(* Schneider Machine Expert - Basic project plc_prog_for_SoMachine_Basic, file version 2.2.0.0 *)
(* CompanyInformations: Name=SmallSystems *)
(* ProjectInformations: Name=Garden Water Control Centre, Description=Lorem ipsum dolor sit amet, consetetur sadipscing elitr, sed diam nonumy eirmod tempor invidunt ut labore et dolore magna aliquyam erat, sed diam voluptua. At vero eos et accusam et justo duo dolores et ea rebum. Stet clita kasd gubergren, no sea takimata sanctus est Lorem ipsum dolor sit amet. Lorem ipsum dolor sit amet, consetetur sadipscing elitr, sed diam nonumy eirmod tempor invidunt ut labore et dolore magna aliquyam erat, sed diam voluptua. At vero eos et accusam et justo duo dolores et ea rebum. Stet clita kasd gubergren, no sea takimata sanctus est Lorem ipsum dolor sit amet. *)
(* UserInformations: LastName=Wilhelm, FirstName=Konstantin, Email=admin@kw.smallsystems.ru, State=Brandenburg, Country=Germany *)

HARDWARE
  Cpu 0: TM221C16R
  EthernetConfiguration: NetworkName=M221, IpAllocationMode=FixedAddress, IpAddress=0.0.0.0, SubnetMask=0.0.0.0
  SerialLineConfiguration: Baud=Baud19200, Parity=ParityEven, DataBits=DataBits8, StopBits=StopBits1, PhysicalMedium=PhysicalMediumRs485, TransmissionMode=TransmissionModeModbusRtu, SlaveId=1, Addressing=SlaveAddressing
  MastTask: UsePeriodScanMode=false, PeriodScan=100
  FastTask: Period=255
  CpuBehavior: StartingMode=StartAsPreviousState, AutoSaveRamOnEeprom=true, WatchdogPeriod=250

SYMBOLS  (address, symbol, comment, settings)
  %M0       P_IN_RELEASE  "Freigabe für die Pumpe"
  %M1       P_IN_DELAY  "bei =1 darf die Pumpe NICHT AN sein"
  %M2       P_IN_TIMEOUT  "bei =1 muss die Pumpe ausgeschaltet sein"
  %M3       P_IN_OVERLOAD  "bei =1 muss die Pumpe ausgeschaltet sein"
  %M4       P_IN_OVERHEAT  "bei =1 muss die Pumpe ausgeschaltet sein"
  %M5       P_IN_BIT  "Merker, der das Status der Pumpe bestimmt"
  %M6       C_PIN_ERROR
  %M7       C_PIN_PRESET
  %M8       C_PIN_RESET
  %M9       C_PIN_SET
  %M10      C_PIN_CD
  %M11      P_OUT_RELEASE
  %M12      P_OUT_DELAY
  %M13      P_OUT_OVERLOAD
  %M14      P_OUT_OVERHEAT
  %M15      P_OUT_BIT
  %M16      P_OUT_TIMEOUT
  %M17      C_POUT_ERROR
  %M18      C_POUT_PRESET
  %M19      C_POUT_RESET
  %M20      C_POUT_SET
  %M21      C_POUT_CD
  %M22      VLV_TNK_UP_LEFT  "EINgangsventil im linken Behälter"
  %M23      VLV_TNK_UP_RIGHT  "EINgangsventil im rechten Behälter"
  %M24      VLV_IN_EXTENTION  "Zusätzlicher Vertil/Hand für Nebenanschluß an Pumpe_IN (Optional)"
  %M25      VLV_TNK_DOWN_LEFT  "AUSgangsventil im linken Behälter"
  %M26      VLV_TNK_DOWN_RIGHT  "AUSgangsventil im rechten Behälter"
  %M27      VLV_OUT_EXTENTION
  %M28      OUT_WITH_PRESSURE
  %M29      HIGH_LVL_TNK_LEFT  "Im linken Behälter hat das Wasser Höhepunk erreicht"
  %M30      HIGH_LVL_TNK_RIGHT  "Im linken Behälter hat das Wasser Höhepunk erreicht"
  %M31      LOW_LVL_TNK_LEFT
  %M32      LOW_LVL_TNK_RIGHT
  %M33      FILL_TNK_LEFT
  %M34      FILL_TNK_RIGHT
  %M35      DRAIN_TNK_LEFT
  %M36      DRAIN_TNK_RIGHT
  %S6       SB_TB1S  "Von einer internen Uhr generierte Zeitbasis 1 s"
  %S13      SB_FIRSTRUN  "Verweist auf den ersten Steuerungszyklus im RUN-Betrieb."
  %MW0      PUMP_DELAY_VALUE  "Die Stillzeit, die nach Ausschalten der Pumpe, eingehalten werden soll"
  %MW1      PUMP_TIMEOUT_VALUE  "Wie lange darf die Pumpe ununterbrochen laufen"
  %TM0      TP_P_IN  "Timer für die Pause zwischen EINschalten der Pumpe"  [Type=TP, Preset=120, Base=OneSecond]
  %TM1      TON_P_IN  "Timer für die maximale Dauer eines Einschltens"  [Preset=1200, Base=OneSecond]
  %TM2      TP_P_OUT  "Timer für die Pause zwischen EINschalten der Pumpe"  [Type=TP, Preset=120, Base=OneSecond]
  %TM3      TON_P_OUT  "Timer für die maximale Dauer eines Einschltens"  [Preset=1200, Base=OneSecond]
  %TM4        [Preset=10, Base=OneSecond]
  %TM5        [Preset=2, Base=OneSecond]
  %TM6        [Preset=2, Base=OneSecond]
  %TM7        [Preset=20, Base=OneSecond]
  %TM8        [Preset=20, Base=OneSecond]
  %TM9        [Preset=20, Base=OneSecond]
  %C0       COUNTER_P_IN  "Zählt die Arbeitszeit in Sekunden"  [Preset=7200]
  %C1       COUNTER_P_OUT  "Zählt die Arbeitszeit in Sekunden"  [Preset=7200]
  %I0.0     I_0_0
  %Q0.0     Q_0_0

POU IO
  (* SectionNumber=1 *)

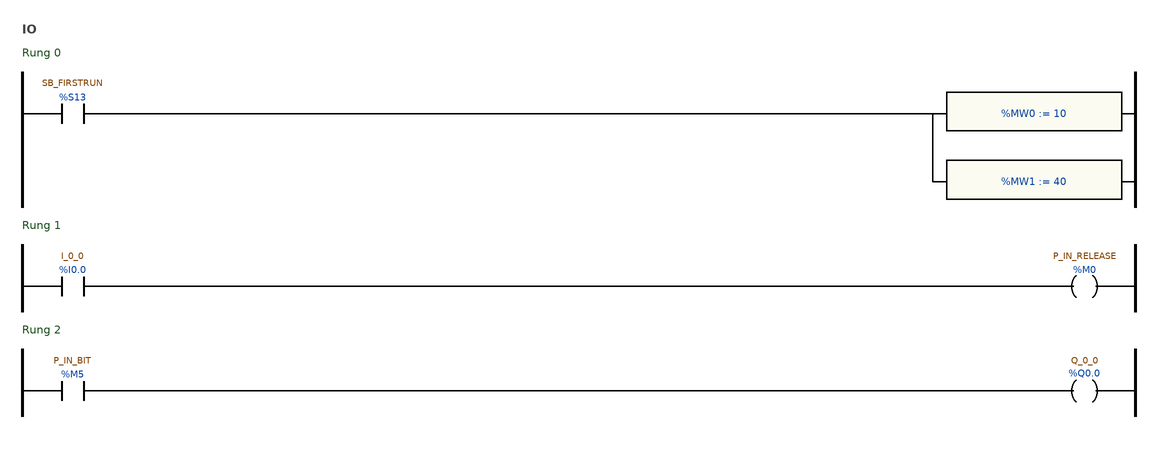

// Rung 0
  LD %S13                 (* SB_FIRSTRUN *)
  [ %MW0 := 10 ]          (* PUMP_DELAY_VALUE *)
  [ %MW1 := 40 ]          (* PUMP_TIMEOUT_VALUE *)
  // as ST:
  //   IF SB_FIRSTRUN THEN PUMP_DELAY_VALUE := 10; END_IF;
  //   IF SB_FIRSTRUN THEN PUMP_TIMEOUT_VALUE := 40; END_IF;

// Rung 1
  LD %I0.0                (* I_0_0 *)
  ST %M0                  (* P_IN_RELEASE *)
  // as ST:
  //   P_IN_RELEASE := I_0_0;

// Rung 2
  LD %M5                  (* P_IN_BIT *)
  ST %Q0.0                (* Q_0_0 *)
  // as ST:
  //   Q_0_0 := P_IN_BIT;

POU Valves
  (* SectionNumber=2 *)

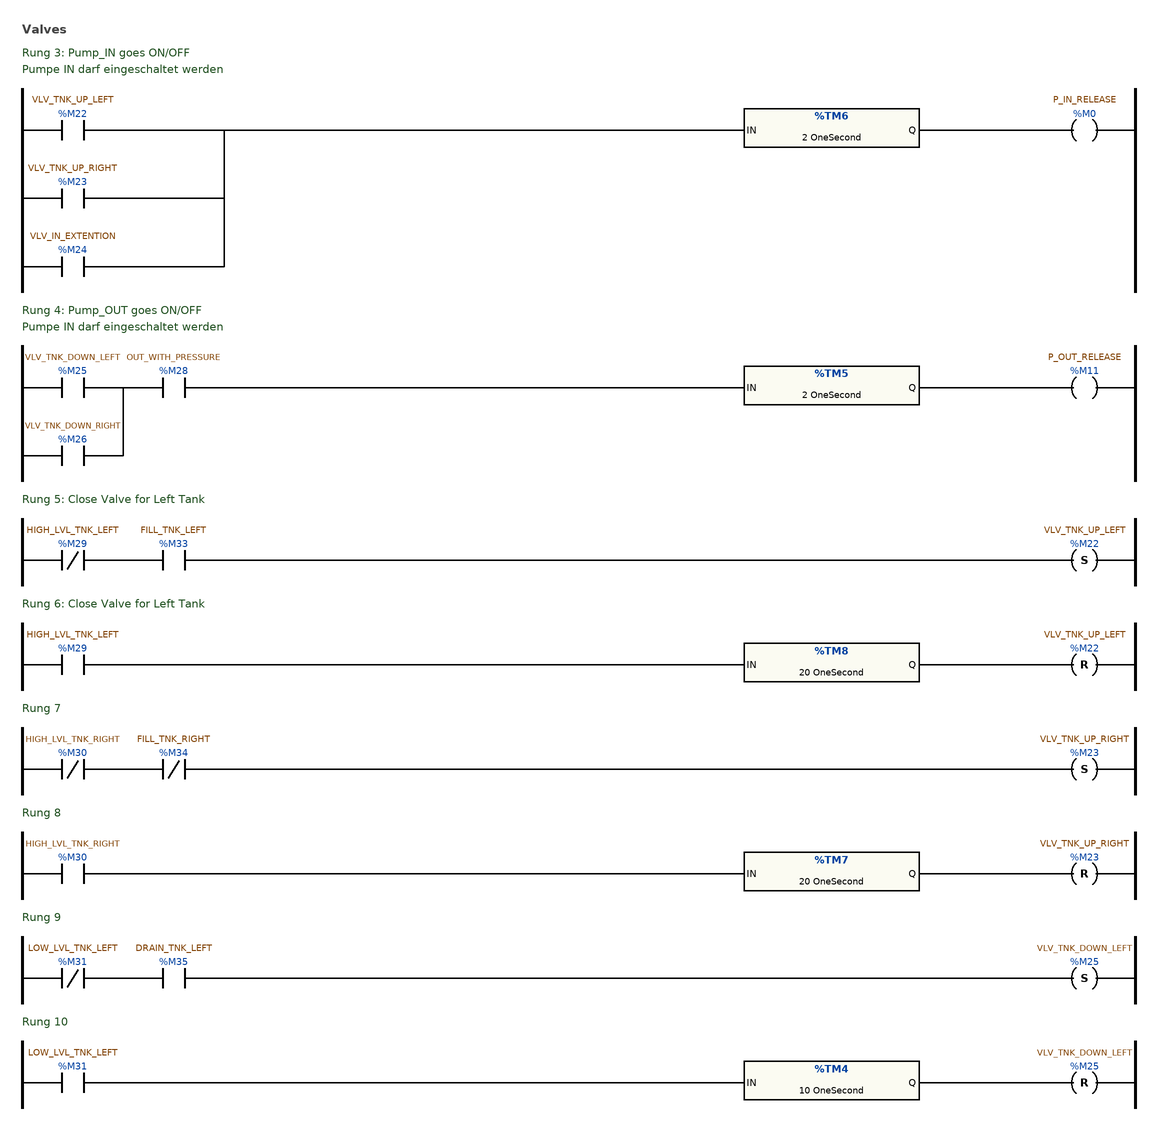

// Rung 3: Pump_IN goes ON/OFF
// Pumpe IN darf eingeschaltet werden
  BLK %TM6
  LD %M22                 (* VLV_TNK_UP_LEFT *)
  OR %M23                 (* VLV_TNK_UP_RIGHT *)
  OR %M24                 (* VLV_IN_EXTENTION *)
  IN
  OUT_BLK
  LD Q
  ST %M0                  (* P_IN_RELEASE *)
  END_BLK
  // as ST:
  //   %TM6(IN := VLV_TNK_UP_LEFT OR VLV_TNK_UP_RIGHT OR VLV_IN_EXTENTION);
  //   P_IN_RELEASE := %TM6.Q;

// Rung 4: Pump_OUT goes ON/OFF
// Pumpe IN darf eingeschaltet werden
  BLK %TM5
  LD %M25                 (* VLV_TNK_DOWN_LEFT *)
  OR %M26                 (* VLV_TNK_DOWN_RIGHT *)
  AND %M28                (* OUT_WITH_PRESSURE *)
  IN
  OUT_BLK
  LD Q
  ST %M11                 (* P_OUT_RELEASE *)
  END_BLK
  // as ST:
  //   %TM5(IN := (VLV_TNK_DOWN_LEFT OR VLV_TNK_DOWN_RIGHT) AND OUT_WITH_PRESSURE);
  //   P_OUT_RELEASE := %TM5.Q;

// Rung 5: Close Valve for Left Tank
  LDN %M29                (* HIGH_LVL_TNK_LEFT *)
  AND %M33                (* FILL_TNK_LEFT *)
  S %M22                  (* VLV_TNK_UP_LEFT *)
  // as ST:
  //   IF NOT HIGH_LVL_TNK_LEFT AND FILL_TNK_LEFT THEN VLV_TNK_UP_LEFT := TRUE; END_IF;

// Rung 6: Close Valve for Left Tank
  BLK %TM8
  LD %M29                 (* HIGH_LVL_TNK_LEFT *)
  IN
  OUT_BLK
  LD Q
  R %M22                  (* VLV_TNK_UP_LEFT *)
  END_BLK
  // as ST:
  //   %TM8(IN := HIGH_LVL_TNK_LEFT);
  //   IF %TM8.Q THEN VLV_TNK_UP_LEFT := FALSE; END_IF;

// Rung 7
  LDN %M30                (* HIGH_LVL_TNK_RIGHT *)
  ANDN %M34               (* FILL_TNK_RIGHT *)
  S %M23                  (* VLV_TNK_UP_RIGHT *)
  // as ST:
  //   IF NOT HIGH_LVL_TNK_RIGHT AND NOT FILL_TNK_RIGHT THEN VLV_TNK_UP_RIGHT := TRUE; END_IF;

// Rung 8
  BLK %TM7
  LD %M30                 (* HIGH_LVL_TNK_RIGHT *)
  IN
  OUT_BLK
  LD Q
  R %M23                  (* VLV_TNK_UP_RIGHT *)
  END_BLK
  // as ST:
  //   %TM7(IN := HIGH_LVL_TNK_RIGHT);
  //   IF %TM7.Q THEN VLV_TNK_UP_RIGHT := FALSE; END_IF;

// Rung 9
  LDN %M31                (* LOW_LVL_TNK_LEFT *)
  AND %M35                (* DRAIN_TNK_LEFT *)
  S %M25                  (* VLV_TNK_DOWN_LEFT *)
  // as ST:
  //   IF NOT LOW_LVL_TNK_LEFT AND DRAIN_TNK_LEFT THEN VLV_TNK_DOWN_LEFT := TRUE; END_IF;

// Rung 10
  BLK %TM4
  LD %M31                 (* LOW_LVL_TNK_LEFT *)
  IN
  OUT_BLK
  LD Q
  R %M25                  (* VLV_TNK_DOWN_LEFT *)
  END_BLK
  // as ST:
  //   %TM4(IN := LOW_LVL_TNK_LEFT);
  //   IF %TM4.Q THEN VLV_TNK_DOWN_LEFT := FALSE; END_IF;

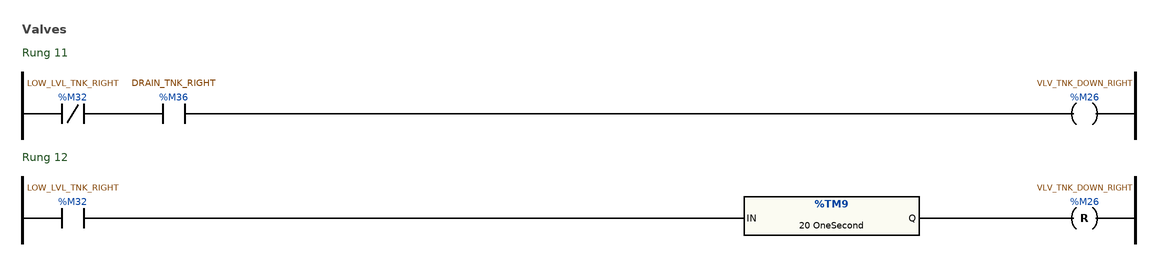

// Rung 11
  LDN %M32                (* LOW_LVL_TNK_RIGHT *)
  AND %M36                (* DRAIN_TNK_RIGHT *)
  ST %M26                 (* VLV_TNK_DOWN_RIGHT *)
  // as ST:
  //   VLV_TNK_DOWN_RIGHT := NOT LOW_LVL_TNK_RIGHT AND DRAIN_TNK_RIGHT;

// Rung 12
  BLK %TM9
  LD %M32                 (* LOW_LVL_TNK_RIGHT *)
  IN
  OUT_BLK
  LD Q
  R %M26                  (* VLV_TNK_DOWN_RIGHT *)
  END_BLK
  // as ST:
  //   %TM9(IN := LOW_LVL_TNK_RIGHT);
  //   IF %TM9.Q THEN VLV_TNK_DOWN_RIGHT := FALSE; END_IF;

POU Pumps
  (* SectionNumber=3 *)

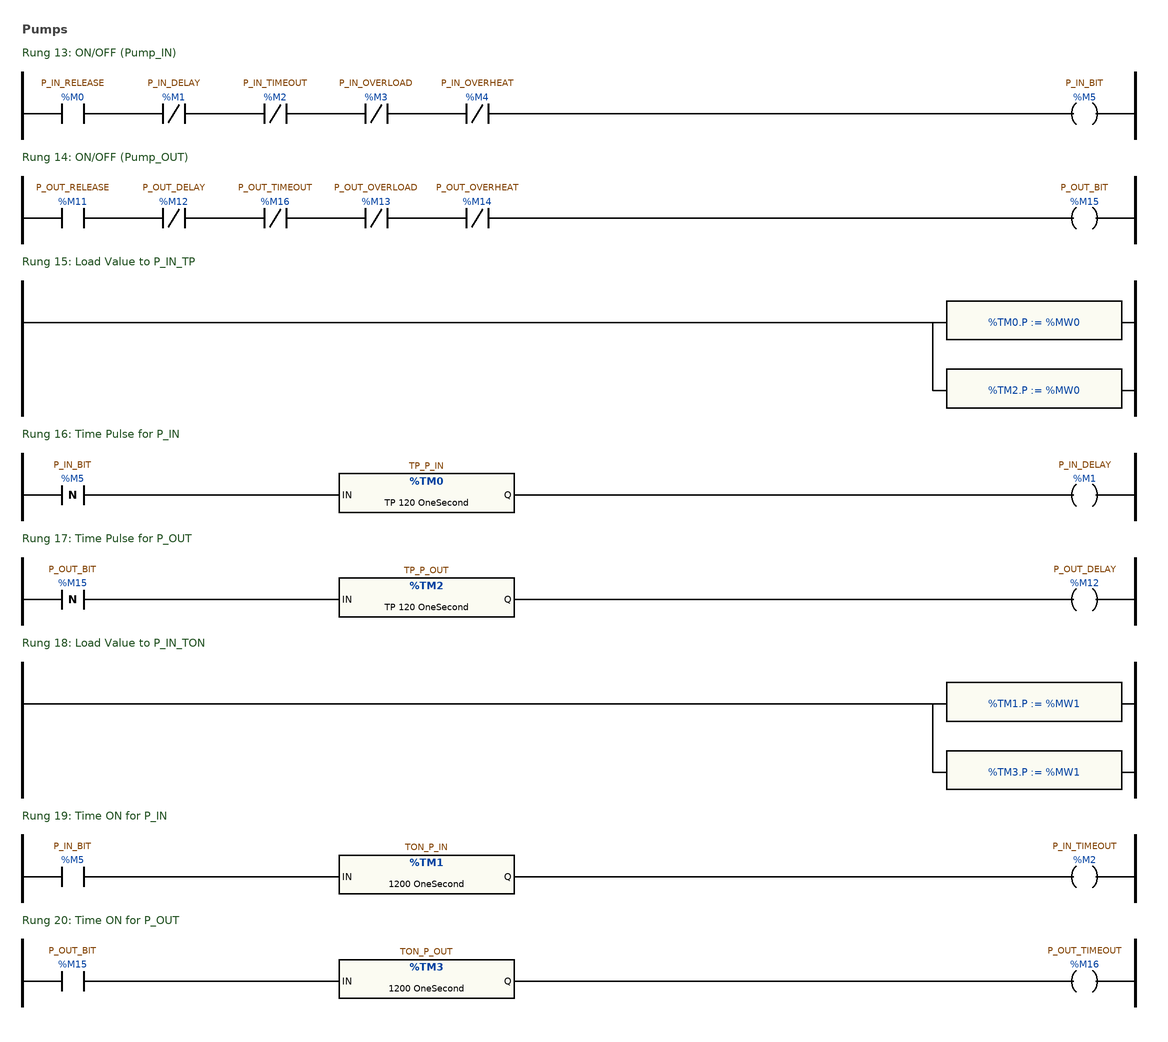

// Rung 13: ON/OFF (Pump_IN)
  LD %M0                  (* P_IN_RELEASE *)
  ANDN %M1                (* P_IN_DELAY *)
  ANDN %M2                (* P_IN_TIMEOUT *)
  ANDN %M3                (* P_IN_OVERLOAD *)
  ANDN %M4                (* P_IN_OVERHEAT *)
  ST %M5                  (* P_IN_BIT *)
  // as ST:
  //   P_IN_BIT := P_IN_RELEASE AND NOT P_IN_DELAY AND NOT P_IN_TIMEOUT AND NOT P_IN_OVERLOAD AND NOT P_IN_OVERHEAT;

// Rung 14: ON/OFF (Pump_OUT)
  LD %M11                 (* P_OUT_RELEASE *)
  ANDN %M12               (* P_OUT_DELAY *)
  ANDN %M16               (* P_OUT_TIMEOUT *)
  ANDN %M13               (* P_OUT_OVERLOAD *)
  ANDN %M14               (* P_OUT_OVERHEAT *)
  ST %M15                 (* P_OUT_BIT *)
  // as ST:
  //   P_OUT_BIT := P_OUT_RELEASE AND NOT P_OUT_DELAY AND NOT P_OUT_TIMEOUT AND NOT P_OUT_OVERLOAD AND NOT P_OUT_OVERHEAT;

// Rung 15: Load Value to P_IN_TP
  LD 1
  [ %TM0.P := %MW0 ]      (* TP_P_IN, PUMP_DELAY_VALUE - Laden Preset des Timers aus der Variable *)
  [ %TM2.P := %MW0 ]      (* TP_P_OUT, PUMP_DELAY_VALUE - Laden Preset des Timers aus der Variable *)
  // as ST:
  //   TP_P_IN.P := PUMP_DELAY_VALUE;
  //   TP_P_OUT.P := PUMP_DELAY_VALUE;

// Rung 16: Time Pulse for P_IN
  BLK %TM0                (* TP_P_IN *)
  LDF %M5                 (* P_IN_BIT *)
  IN
  OUT_BLK
  LD Q
  ST %M1                  (* P_IN_DELAY *)
  END_BLK
  // as ST:
  //   TP_P_IN(IN := FALLING(P_IN_BIT));
  //   P_IN_DELAY := TP_P_IN.Q;

// Rung 17: Time Pulse for P_OUT
  BLK %TM2                (* TP_P_OUT *)
  LDF %M15                (* P_OUT_BIT *)
  IN
  OUT_BLK
  LD Q
  ST %M12                 (* P_OUT_DELAY *)
  END_BLK
  // as ST:
  //   TP_P_OUT(IN := FALLING(P_OUT_BIT));
  //   P_OUT_DELAY := TP_P_OUT.Q;

// Rung 18: Load Value to P_IN_TON
  LD 1
  [ %TM1.P := %MW1 ]      (* TON_P_IN, PUMP_TIMEOUT_VALUE - Laden Preset des Timers aus der Variable *)
  [ %TM3.P := %MW1 ]      (* TON_P_OUT, PUMP_TIMEOUT_VALUE - Laden Preset des Timers aus der Variable *)
  // as ST:
  //   TON_P_IN.P := PUMP_TIMEOUT_VALUE;
  //   TON_P_OUT.P := PUMP_TIMEOUT_VALUE;

// Rung 19: Time ON for P_IN
  BLK %TM1                (* TON_P_IN *)
  LD %M5                  (* P_IN_BIT *)
  IN
  OUT_BLK
  LD Q
  ST %M2                  (* P_IN_TIMEOUT *)
  END_BLK
  // as ST:
  //   TON_P_IN(IN := P_IN_BIT);
  //   P_IN_TIMEOUT := TON_P_IN.Q;

// Rung 20: Time ON for P_OUT
  BLK %TM3                (* TON_P_OUT *)
  LD %M15                 (* P_OUT_BIT *)
  IN
  OUT_BLK
  LD Q
  ST %M16                 (* P_OUT_TIMEOUT *)
  END_BLK
  // as ST:
  //   TON_P_OUT(IN := P_OUT_BIT);
  //   P_OUT_TIMEOUT := TON_P_OUT.Q;

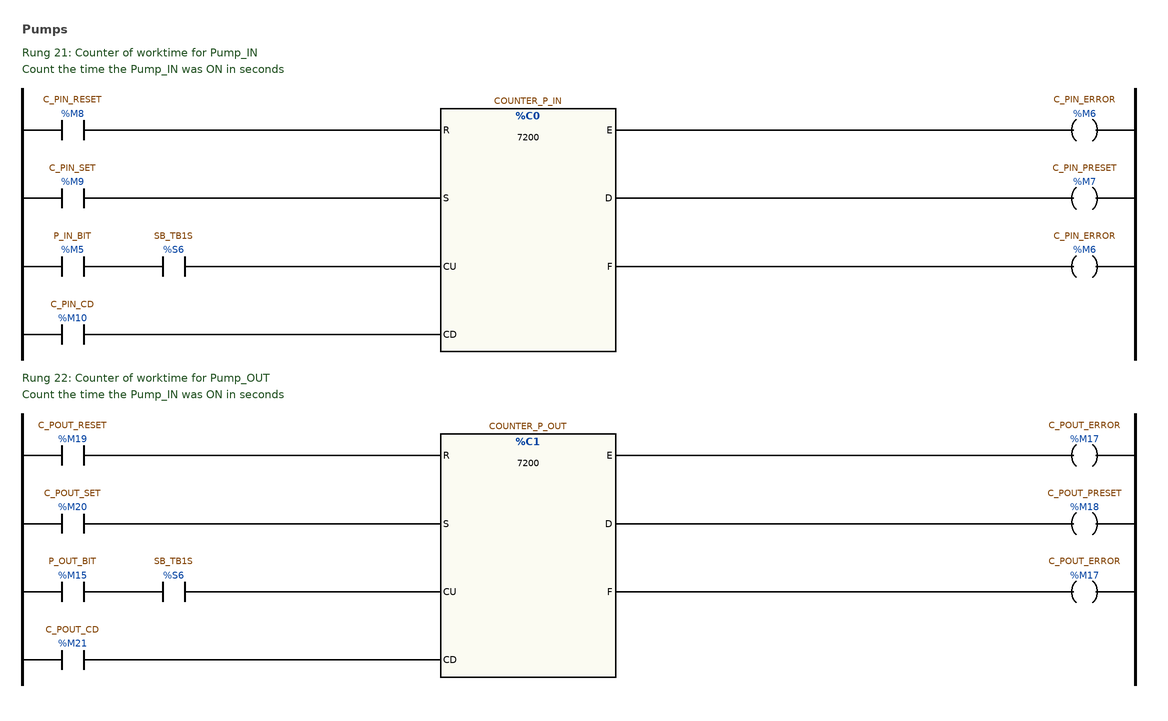

// Rung 21: Counter of worktime for Pump_IN
// Count the time the Pump_IN was ON in seconds
  BLK %C0                 (* COUNTER_P_IN *)
  LD %M8                  (* C_PIN_RESET *)
  R
  LD %M9                  (* C_PIN_SET *)
  S
  LD %M5                  (* P_IN_BIT *)
  AND %S6                 (* SB_TB1S *)
  CU
  LD %M10                 (* C_PIN_CD *)
  CD
  OUT_BLK
  LD E
  ST %M6                  (* C_PIN_ERROR *)
  LD D
  ST %M7                  (* C_PIN_PRESET *)
  LD F
  ST %M6                  (* C_PIN_ERROR *)
  END_BLK
  // as ST:
  //   COUNTER_P_IN(R := C_PIN_RESET, S := C_PIN_SET, CU := P_IN_BIT AND SB_TB1S, CD := C_PIN_CD);
  //   C_PIN_ERROR := COUNTER_P_IN.E;
  //   C_PIN_PRESET := COUNTER_P_IN.D;
  //   C_PIN_ERROR := COUNTER_P_IN.F;

// Rung 22: Counter of worktime for Pump_OUT
// Count the time the Pump_IN was ON in seconds
  BLK %C1                 (* COUNTER_P_OUT *)
  LD %M19                 (* C_POUT_RESET *)
  R
  LD %M20                 (* C_POUT_SET *)
  S
  LD %M15                 (* P_OUT_BIT *)
  AND %S6                 (* SB_TB1S *)
  CU
  LD %M21                 (* C_POUT_CD *)
  CD
  OUT_BLK
  LD E
  ST %M17                 (* C_POUT_ERROR *)
  LD D
  ST %M18                 (* C_POUT_PRESET *)
  LD F
  ST %M17                 (* C_POUT_ERROR *)
  END_BLK
  // as ST:
  //   COUNTER_P_OUT(R := C_POUT_RESET, S := C_POUT_SET, CU := P_OUT_BIT AND SB_TB1S, CD := C_POUT_CD);
  //   C_POUT_ERROR := COUNTER_P_OUT.E;
  //   C_POUT_PRESET := COUNTER_P_OUT.D;
  //   C_POUT_ERROR := COUNTER_P_OUT.F;
